{attribute 'linkalways'} 
{attribute 'no_explicit_call' := 'This FB is a CLASS and must be accessed using methods or properties'}
{attribute 'enable_dynamic_creation'}
FUNCTION_BLOCK JsonSerializer EXTENDS Disposable IMPLEMENTS I_Serializer;
VAR
	jsonSaxWriter : FB_JsonSaxWriter;
END_VAR

METHOD PUBLIC AddBase64 : I_Serializer
VAR_INPUT
	pBytes : POINTER TO BYTE;
	nBytes : DINT;
END_VAR
jsonSaxWriter.AddBase64(pBytes, nBytes);
AddBase64 := THIS^;
END_METHOD

METHOD PUBLIC AddBool : I_Serializer
VAR_INPUT
	Value : BOOL;
END_VAR
jsonSaxWriter.AddBool(Value);
AddBool := THIS^;
END_METHOD

METHOD PUBLIC AddByte : I_Serializer
VAR_INPUT
	Value : BYTE;
END_VAR
jsonSaxWriter.AddUDint(BYTE_TO_UDINT(Value));
AddByte := THIS^;
END_METHOD

METHOD PUBLIC AddBytesAsHex : I_Serializer
VAR_INPUT
	pBytes : POINTER TO BYTE;
	nBytes : DINT;
END_VAR
jsonSaxWriter.AddHexBinary(pBytes, nBytes);
AddBytesAsHex := THIS^;
END_METHOD

METHOD PUBLIC AddDateTime : I_Serializer
VAR_INPUT
	Value : DATE_AND_TIME;
END_VAR
jsonSaxWriter.AddDateTime(Value);
AddDateTime := THIS^;
END_METHOD

METHOD PUBLIC AddDcTime : I_Serializer
VAR_INPUT
	Value : DCTIME;
END_VAR
jsonSaxWriter.AddDcTime(Value);
AddDcTime := THIS^;
END_METHOD

METHOD PUBLIC AddDint : I_Serializer
VAR_INPUT
	Value : DINT;
END_VAR
jsonSaxWriter.AddDint(Value);
AddDint := THIS^;
END_METHOD

METHOD PUBLIC AddDword : I_Serializer
VAR_INPUT
	Value : DWORD;
END_VAR
jsonSaxWriter.AddUDint(DWORD_TO_UDINT(Value));
AddDword := THIS^;
END_METHOD

METHOD PUBLIC AddFileTime : I_Serializer
VAR_INPUT
	Value : FILETIME;
END_VAR
jsonSaxWriter.AddFileTime(Value);
AddFileTime := THIS^;
END_METHOD

METHOD PUBLIC AddInt : I_Serializer
VAR_INPUT
	Value : INT;
END_VAR
jsonSaxWriter.AddDint(INT_TO_DINT(Value));
AddInt := THIS^;
END_METHOD

METHOD PUBLIC AddKey : I_Serializer
VAR_INPUT
	Key : T_MAXSTRING;
END_VAR
jsonSaxWriter.AddKey(Key);
AddKey := THIS^;
END_METHOD

METHOD PUBLIC AddKeyBase64 : I_Serializer
VAR_INPUT
	Key : T_MAXSTRING;
	pBytes : POINTER TO BYTE;
	nBytes : DINT;
END_VAR
AddKey(Key);
AddBase64(pBytes, nBytes);
AddKeyBase64 := THIS^;
END_METHOD

METHOD PUBLIC AddKeyBool : I_Serializer
VAR_INPUT
	Key : T_MAXSTRING;
	Value : BOOL;
END_VAR
AddKey(Key);
AddBool(Value);
AddKeyBool := THIS^;
END_METHOD

METHOD PUBLIC AddKeyByte : I_Serializer
VAR_INPUT
	Key : T_MAXSTRING;
	Value : BYTE;
END_VAR
AddKey(Key);
AddByte(Value);
AddKeyByte := THIS^;
END_METHOD

METHOD PUBLIC AddKeyBytesAsHex : I_Serializer
VAR_INPUT
	Key : T_MAXSTRING;
	pBytes : POINTER TO BYTE;
	nBytes : DINT;
END_VAR
AddKey(Key);
AddBytesAsHex(pBytes, nBytes);
AddKeyBytesAsHex := THIS^;
END_METHOD

METHOD PUBLIC AddKeyDateTime : I_Serializer
VAR_INPUT
	Key : T_MAXSTRING;
	Value : DATE_AND_TIME;
END_VAR
AddKey(Key);
AddDateTime(Value);
AddKeyDateTime := THIS^;
END_METHOD

METHOD PUBLIC AddKeyDcTime : I_Serializer
VAR_INPUT
	Key : T_MAXSTRING;
	Value : DCTIME;
END_VAR
AddKey(Key);
AddDcTime(Value);
AddKeyDcTime := THIS^;
END_METHOD

METHOD PUBLIC AddKeyDint : I_Serializer
VAR_INPUT
	Key : T_MAXSTRING;
	Value : DINT;
END_VAR
AddKey(Key);
AddDint(Value);
AddKeyDint := THIS^;
END_METHOD

METHOD PUBLIC AddKeyDword : I_Serializer
VAR_INPUT
	Key : T_MAXSTRING;
	Value : DWORD;
END_VAR
AddKey(Key);
AddDword(Value);
AddKeyDword := THIS^;
END_METHOD

METHOD PUBLIC AddKeyFileTime : I_Serializer
VAR_INPUT
	Key : T_MAXSTRING;
	Value : FILETIME;
END_VAR
AddKey(Key);
AddFileTime(Value);
AddKeyFileTime := THIS^;
END_METHOD

METHOD PUBLIC AddKeyInt : I_Serializer
VAR_INPUT
	Key : T_MAXSTRING;
	Value : INT;
END_VAR
AddKey(Key);
AddInt(Value);
AddKeyInt := THIS^;
END_METHOD

METHOD PUBLIC AddKeyLint : I_Serializer
VAR_INPUT
	Key : T_MAXSTRING;
	Value : LINT;
END_VAR
AddKey(Key);
AddLint(Value);
AddKeyLint := THIS^;
END_METHOD

METHOD PUBLIC AddKeyLreal : I_Serializer
VAR_INPUT
	Key : T_MAXSTRING;
	Value : LREAL;
END_VAR
AddKey(Key);
AddLreal(Value);
AddKeyLreal := THIS^;
END_METHOD

METHOD PUBLIC AddKeyLtime : I_Serializer
VAR_INPUT
	Key : T_MAXSTRING;
	Value : LTIME;
END_VAR
AddKey(Key);
AddLTIME(Value);
AddKeyLtime := THIS^;
END_METHOD

METHOD PUBLIC AddKeyLword : I_Serializer
VAR_INPUT
	Key : T_MAXSTRING;
	Value : LWORD;
END_VAR
AddKey(Key);
AddLword(Value);
AddKeyLword := THIS^;
END_METHOD

METHOD PUBLIC AddKeyNull : I_Serializer
VAR_INPUT
	Key : T_MAXSTRING;
END_VAR
AddKey(Key);
AddNull();
AddKeyNull := THIS^;
END_METHOD

METHOD PUBLIC AddKeyObject : I_Serializer
VAR_INPUT
	Key : T_MAXSTRING;
	Object : I_Serializable;
END_VAR
AddKey(Key);
Object.SerializeWith(THIS^);
AddKeyObject := THIS^;
END_METHOD

METHOD PUBLIC AddKeyRawJson : I_Serializer
VAR_INPUT
	Key : T_MAXSTRING;
	RawObject : REFERENCE TO STRING;;
END_VAR
AddKey(Key);
AddRawJson(RawObject);
AddKeyRawJson := THIS^;
END_METHOD

METHOD PUBLIC AddKeyReal : I_Serializer
VAR_INPUT
	Key : T_MAXSTRING;
	Value : REAL;
END_VAR
AddKey(Key);
AddReal(Value);
AddKeyReal := THIS^;
END_METHOD

METHOD PUBLIC AddKeySint : I_Serializer
VAR_INPUT
	Key : T_MAXSTRING;
	Value : SINT;
END_VAR
AddKey(Key);
AddSint(Value);
AddKeySint := THIS^;
END_METHOD

METHOD PUBLIC AddKeyString : I_Serializer
VAR_INPUT
	Key : T_MAXSTRING;
	Value : T_MAXSTRING;
END_VAR
AddKey(Key);
AddString(Value);
AddKeyString := THIS^;
END_METHOD

METHOD PUBLIC AddKeyStringByRef : I_Serializer
VAR_INPUT
	Key : T_MAXSTRING;
	Value : REFERENCE TO STRING;;
END_VAR
AddKey(Key);
AddStringByRef(Value);
AddKeyStringByRef := THIS^;
END_METHOD

METHOD PUBLIC AddKeyTime : I_Serializer
VAR_INPUT
	Key : T_MAXSTRING;
	Value : TIME;
END_VAR
AddKey(Key);
AddTime(Value);
AddKeyTime := THIS^;
END_METHOD

METHOD PUBLIC AddKeyTod : I_Serializer
VAR_INPUT
	Key : T_MAXSTRING;
	Value : TOD;
END_VAR
AddKey(Key);
AddTod(Value);
AddKeyTod := THIS^;
END_METHOD

METHOD PUBLIC AddKeyUdint : I_Serializer
VAR_INPUT
	Key : T_MAXSTRING;
	Value : UDINT;
END_VAR
AddKey(Key);
AddUdint(Value);
AddKeyUdint := THIS^;
END_METHOD

METHOD PUBLIC AddKeyUint : I_Serializer
VAR_INPUT
	Key : T_MAXSTRING;
	Value : UINT;
END_VAR
AddKey(Key);
AddUint(Value);
AddKeyUint := THIS^;
END_METHOD

METHOD PUBLIC AddKeyUlint : I_Serializer
VAR_INPUT
	Key : T_MAXSTRING;
	Value : ULINT;
END_VAR
AddKey(Key);
AddUlint(Value);
AddKeyUlint := THIS^;
END_METHOD

METHOD PUBLIC AddKeyUsint : I_Serializer
VAR_INPUT
	Key : T_MAXSTRING;
	Value : USINT;
END_VAR
AddKey(Key);
AddUsint(Value);
AddKeyUsint := THIS^;
END_METHOD

METHOD PUBLIC AddKeyWord : I_Serializer
VAR_INPUT
	Key : T_MAXSTRING;
	Value : WORD;
END_VAR
AddKey(Key);
AddWord(Value);
AddKeyWord := THIS^;
END_METHOD

METHOD PUBLIC AddLint : I_Serializer
VAR_INPUT
	Value : LINT;
END_VAR
jsonSaxWriter.AddLint(Value);
AddLint := THIS^;
END_METHOD

METHOD PUBLIC AddLreal : I_Serializer
VAR_INPUT
	Value : LREAL;
END_VAR
jsonSaxWriter.AddLreal(Value);
AddLreal := THIS^;
END_METHOD

METHOD PUBLIC AddLtime : I_Serializer
VAR_INPUT
	Value : LTIME;
END_VAR
VAR
	converted : T_MAXSTRING;
END_VAR
converted := LTIME_TO_STRING(Value);
jsonSaxWriter.AddString(converted);
AddLtime := THIS^;
END_METHOD

METHOD PUBLIC AddLword : I_Serializer
VAR_INPUT
	Value : LWORD;
END_VAR
jsonSaxWriter.AddUlint(LWORD_TO_ULINT(Value));
AddLword := THIS^;
END_METHOD

METHOD PUBLIC AddNull : I_Serializer
VAR_INPUT
END_VAR
jsonSaxWriter.AddNull();
AddNull := THIS^;
END_METHOD

METHOD PUBLIC AddObject
VAR_INPUT
	Object : I_Serializable;
END_VAR
Object.SerializeWith(This^);
END_METHOD

METHOD PUBLIC AddRawJson
VAR_INPUT
	RawObject : REFERENCE TO STRING;
END_VAR
jsonSaxWriter.AddRawObject(RawObject);
END_METHOD

METHOD PUBLIC AddReal : I_Serializer
VAR_INPUT
	Value : REAL;
END_VAR
// real to lreal is used to negate an issue with TC4024.55 which prevents max REAL from being serailized.  
// so a REAL_TO_LREAL conversion is made to ensure this is always possible.  
jsonSaxWriter.AddLReal(REAL_TO_LREAL(Value));
AddReal := THIS^;
END_METHOD

METHOD PUBLIC AddSint : I_Serializer
VAR_INPUT
	Value : SINT;
END_VAR
jsonSaxWriter.AddDint(SINT_TO_DINT(Value));
AddSint := THIS^;
END_METHOD

METHOD PUBLIC AddString : I_Serializer
VAR_INPUT
	Value : T_MAXSTRING;
END_VAR
jsonSaxWriter.AddString(Value);
AddString := THIS^;
END_METHOD

METHOD PUBLIC AddStringByRef : I_Serializer
VAR_INPUT
	Value : REFERENCE TO STRING;
END_VAR
jsonSaxWriter.AddString(Value);
AddStringByRef := THIS^;
END_METHOD

METHOD PUBLIC AddTime : I_Serializer
VAR_INPUT
	Value : TIME;
END_VAR
VAR
	converted : T_MAXSTRING;
END_VAR
converted := TIME_TO_STRING(Value);
jsonSaxWriter.AddString(converted);
AddTime := THIS^;
END_METHOD

METHOD PUBLIC AddTod : I_Serializer
VAR_INPUT
	Value : TOD;
END_VAR
VAR
	converted : T_MAXSTRING;
END_VAR
converted := TOD_TO_STRING(Value);
jsonSaxWriter.AddString(converted);
AddTod := THIS^;
END_METHOD

METHOD PUBLIC AddUdint : I_Serializer
VAR_INPUT
	Value : UDINT;
END_VAR
jsonSaxWriter.AddUdint(Value);
AddUdint := THIS^;
END_METHOD

METHOD PUBLIC AddUint : I_Serializer
VAR_INPUT
	Value : UINT;
END_VAR
jsonSaxWriter.AddDint(UINT_TO_DINT(Value));
AddUint := THIS^;
END_METHOD

METHOD PUBLIC AddUlint : I_Serializer
VAR_INPUT
	Value : ULINT;
END_VAR
jsonSaxWriter.AddUlint(Value);
AddUlint := THIS^;
END_METHOD

METHOD PUBLIC AddUsint : I_Serializer
VAR_INPUT
	Value : USINT;
END_VAR
jsonSaxWriter.AddDint(USINT_TO_DINT(Value));
AddUsint := THIS^;
END_METHOD

METHOD PUBLIC AddWord : I_Serializer
VAR_INPUT
	Value : WORD;
END_VAR
jsonSaxWriter.AddUDint(WORD_TO_UDINT(Value));
AddWord := THIS^;
END_METHOD

METHOD PUBLIC Clone : I_Serializer
VAR
	pClone : POINTER TO JsonSerializer;
	jsonSize : UDINT;
	pJsonString : POINTER TO STRING;
END_VAR
pClone := __NEW(JsonSerializer);
Clone := pClone^;

jsonSize := jsonSaxWriter.GetDocumentLength();

IF jsonSize = 0 THEN
	// no further cloning to do. 
	RETURN;
END_IF

pJsonString := __NEW(BYTE, jsonSize);

IF jsonSaxWriter.CopyDocument(pJsonString^, jsonSize) = 0 THEN
	__DELETE(pJsonString);
	RETURN;
END_IF

pClone^.AddRawJson(pJsonString^);
__DELETE(pJsonString);
END_METHOD

METHOD PUBLIC EndArray : I_Serializer
VAR_INPUT
END_VAR
jsonSaxWriter.EndArray();
EndArray := THIS^;
END_METHOD

METHOD PUBLIC EndObject : I_Serializer
VAR_INPUT
END_VAR
jsonSaxWriter.EndObject();
EndObject := THIS^;
END_METHOD

METHOD FB_exit : BOOL
VAR_INPUT
	bInCopyCode : BOOL; // if TRUE, the exit method is called for exiting an instance that is copied afterwards (online change).
END_VAR
IF bInCopyCode THEN
	RETURN;
END_IF

jsonSaxWriter.ResetDocument();
END_METHOD

METHOD PUBLIC GetSerializedDataLength : UDINT
VAR_INPUT
END_VAR
GetSerializedDataLength := jsonSaxWriter.GetDocumentLength();
END_METHOD

METHOD PUBLIC Reset
VAR_INPUT
END_VAR
jsonSaxWriter.ResetDocument();
END_METHOD

METHOD PUBLIC StartArray : I_Serializer
VAR_INPUT
END_VAR
jsonSaxWriter.StartArray();
StartArray := THIS^;
END_METHOD

METHOD PUBLIC StartObject : I_Serializer
VAR_INPUT
END_VAR
jsonSaxWriter.StartObject();
StartObject := THIS^;
END_METHOD

METHOD TryCopySerializedData : BOOL
VAR_INPUT
	DestinationAddress : PVOID;
	DestinationSize : UDINT;
END_VAR
VAR
	pString : POINTER TO STRING;
END_VAR
pString := DestinationAddress;
TryCopySerializedData := jsonSaxWriter.CopyDocument(pString^, DestinationSize) > 0;
END_METHOD

METHOD TryGetSerializedData : BOOL
VAR_INPUT
	DestinationAddress : PVOID;
	DestinationSize : UDINT;
END_VAR
VAR
	pString : POINTER TO STRING;
END_VAR
pString := DestinationAddress;

IF jsonSaxWriter.CopyDocument(pString^, DestinationSize) = 0 THEN
	RETURN;
END_IF

jsonSaxWriter.ResetDocument();
TryGetSerializedData := TRUE;
END_METHOD

END_FUNCTION_BLOCK

(* stored: Version 1.1.0.1, ProductVersion 3.1.4024.12
   POU JsonSerializer: Id {3a129ab2-a3ab-0899-3d54-0101de2c58bf}, SpecialFunc None
   Folder Destructor: Id {a36d3cd1-d9ba-0f02-223d-25cdbead5310}
   Method AddBase64: Id {37e0cdf8-c8d5-0656-00b5-4796987db7e6}
   Method AddBool: Id {f7faf026-5161-0b38-0388-99e9e46f19bf}
   Method AddByte: Id {e0a31f86-bb64-42a7-88cc-4168cbd65908}
   Method AddBytesAsHex: Id {9c6ac6f1-bd6f-0fa6-224c-14efbda1fcfb}
   Method AddDateTime: Id {1614e7d4-6921-0c29-0fce-5ed9d0952178}
   Method AddDcTime: Id {50e483fa-2281-0872-3d74-ba8568f46015}
   Method AddDint: Id {87e576c5-8da8-0219-1f12-07d66db7ed43}
   Method AddDword: Id {b0881de0-e384-4af7-a20c-6df98d7ad39a}
   Method AddFileTime: Id {1cc6f523-1004-023f-04b9-23aa487a5caf}
   Method AddInt: Id {c0a5b091-0f29-4132-888d-8100689d37a9}
   Method AddKey: Id {5802a444-d5f8-0aef-3aed-4223315ad0fa}
   Method AddKeyBase64: Id {b80780c4-bb70-016d-1857-4c80b5b4a8c5}
   Method AddKeyBool: Id {7c7fedb3-201a-005f-2d12-8aa0f2d08798}
   Method AddKeyByte: Id {1be2bd2f-7a1f-48e4-b1f9-bd65cab7c91d}
   Method AddKeyBytesAsHex: Id {8d5e651a-17e3-0e35-3329-ec5b4fbcc7f4}
   Method AddKeyDateTime: Id {c3f54418-ef77-0b7f-2df0-333e36640fc4}
   Method AddKeyDcTime: Id {86181f80-3d38-087a-05e6-15d9ba7d3cf5}
   Method AddKeyDint: Id {6d098a07-2621-0d46-3562-2fb33d7c07bf}
   Method AddKeyDword: Id {ce60440d-ff44-4333-b0ff-e44d2501e832}
   Method AddKeyFileTime: Id {84e6800f-a464-03ae-32c7-890d6e13bd78}
   Method AddKeyInt: Id {596cb93b-c77e-4ae1-92c6-42e9047b850f}
   Method AddKeyLint: Id {09ce8c7e-f77d-0699-0a80-4e41d415a76f}
   Method AddKeyLreal: Id {a78201b7-f28d-0deb-3f37-cb746f15e130}
   Method AddKeyLtime: Id {d9b6ef96-3a27-4aec-8fe7-cd941c752bfe}
   Method AddKeyLword: Id {6c610c6e-d7ab-45b1-84aa-4f4d7b47d4dc}
   Method AddKeyNull: Id {a8618a9d-6876-09ac-2754-39b9d7474928}
   Method AddKeyObject: Id {e777ba6a-6029-4ba4-8bc9-676d1d60c408}
   Method AddKeyRawJson: Id {6c9dd62a-e5cd-472f-a750-5a146e2ef059}
   Method AddKeyReal: Id {0aea5d26-0d31-0678-0113-468250cbf0eb}
   Method AddKeySint: Id {b28d2dee-26a8-4738-ad0b-6cb2f273fcc5}
   Method AddKeyString: Id {51db4e0c-01a6-45f5-9e37-80deacaeb95c}
   Method AddKeyStringByRef: Id {b004894c-c08c-017f-0632-4659be4bd25b}
   Method AddKeyTime: Id {82e35745-2d3e-4a43-bb35-f554e1baab5b}
   Method AddKeyTod: Id {bd01d365-ebb1-414d-9449-e44d4cc3b565}
   Method AddKeyUdint: Id {858d8f12-c4f3-02f8-147d-9f166bc862a1}
   Method AddKeyUint: Id {e71f11cc-fa25-4311-911b-af1d1d836da1}
   Method AddKeyUlint: Id {ab5719a8-f52b-0b24-2e69-6377d1c57be3}
   Method AddKeyUsint: Id {0cbfced3-dde0-4614-85b6-5dbcee9df675}
   Method AddKeyWord: Id {7ac6ab69-856f-414b-bf20-91795f951e14}
   Method AddLint: Id {6c6d485d-a46d-0db8-06e0-9f6704acdae1}
   Method AddLreal: Id {51213ad5-839c-0aaf-22eb-440baa4436c3}
   Method AddLtime: Id {1ba4acde-e210-4502-ba4a-fd1670d24712}
   Method AddLword: Id {2a356460-54bd-49e2-87ff-8a8dd8de321f}
   Method AddNull: Id {bf9cbdfd-2186-0652-3b0f-04135b7771f6}
   Method AddObject: Id {169b7edb-8088-40d6-a167-766a9d4aefc7}
   Method AddRawJson: Id {89de6b51-c765-0b3f-3e8f-ab641bcee924}
   Method AddReal: Id {427cd8af-a9c8-03a3-170e-85035b900a14}
   Method AddSint: Id {0b5fe11f-8201-4371-854a-a085e158bd7e}
   Method AddString: Id {7b10fa03-7fd0-4983-9f3b-5ee38cf9439a}
   Method AddStringByRef: Id {f50eba30-bfd4-06c0-1d25-7314e9fc4b9d}
   Method AddTime: Id {71f12a02-62be-4dd8-890f-158c282eef3c}
   Method AddTod: Id {1877b285-6b05-48fc-a5a0-1d724ef40174}
   Method AddUdint: Id {a7b6a5c4-af8d-0a71-3b80-c10f04bd9d2c}
   Method AddUint: Id {8aeea217-5899-4e4e-8960-7406e6f692a9}
   Method AddUlint: Id {9d35d897-a889-051e-340f-8887d761e0d5}
   Method AddUsint: Id {c968c0ce-7d22-4034-bed7-aeffab9a22f3}
   Method AddWord: Id {5d7b074c-d8ee-40ee-a9a7-8efcc66454ac}
   Method Clone: Id {5f7680c8-2f5d-079d-16b4-6eb697fa9dfc}
   Method EndArray: Id {9be1f4a4-0b7c-0fe9-1c95-32d20ffd88ae}
   Method EndObject: Id {02efe1dc-1946-0426-2c0b-856f82e57bcd}
   Method FB_exit: Id {a6d92505-8110-0349-2b60-ae5f95550d6a}
   Method GetSerializedDataLength: Id {8612fad9-78b9-0595-0070-8a5f446df6af}
   Method Reset: Id {5f0b5871-a99e-0e83-0c7f-334b84692fb8}
   Method StartArray: Id {ce542d61-ae8f-0547-3923-e87d4d81250b}
   Method StartObject: Id {7c46a59a-e687-0359-204a-c4befe2b6536}
   Method TryCopySerializedData: Id {adad71b4-2e1e-02f8-26de-da80ce054965}
   Method TryGetSerializedData: Id {d6651d2e-c410-0e76-0d0b-492f5c41ee4d} *)
